{attribute 'qualified_only'}
{attribute 'to_string'}
// ------------------------------------------------------------------------- 
//  SRCI Robot Library                                                
// ------------------------------------------------------------------------- 
//                                                                           
//  Object:      SyncReaction                                       
//  Author:      Thorsten Brach                                                
//  Date:        2024-06-01
//
//  Description:                                              
//   
//                                                                           
//  Copyright: 
//    (C) 2024 Thorsten Brach. All rights reserved                                                                                                                                            
//             Licensed under the MIT License.
//                                                                           
//  Disclaimer:                                                                           
//    This project is provided without any guarantee and can be used for   
//    private and commercial purposes. Any use is at the user’s 
//    own risk and responsibility.
//
// -------------------------------------------------------------------------
TYPE SyncReaction :
(
  /// • System behavior unaffected
  NO_REACTION := 0,
  /// • No automatic disable
  /// • Reaction will only apply when RA is disabled
  /// • RA can only be enabled if client and server are synchronized
  NO_AUTOMATIC_DISABLE := 1,  
  /// • No automatic disable
  /// • RA can only be enabled if client and server are synchronized
  /// • RA sequence state will change to interrupted when no command is buffered in the active sequence
  /// • Continuation is only possible if client and server are synchronized
  INTERRUPT_WHEN_SEQUENCE_IS_EMPTY := 2,  
  /// • No automatic disable
  /// • RA can only be enabled if client and server are synchronized
  /// • RA sequence state will change to interrupted
  /// • Continuation is only possible if client and server are synchronized
  IMMEDIATE_INTERRUPT := 3
)USINT;
END_TYPE

{attribute 'qualified_only'}
{attribute 'to_string'}
// ------------------------------------------------------------------------- 
//  SRCI Robot Library                                                
// ------------------------------------------------------------------------- 
//                                                                           
//  Object:      SyncTime                                       
//  Author:      Thorsten Brach                                                
//  Date:        2025-04-13
//
//  Description:                                              
//   
//                                                                           
//  Copyright: 
//    (C) 2025 Thorsten Brach. All rights reserved                                                                                                                                            
//             Licensed under the MIT License.
//                                                                           
//  Disclaimer:                                                                           
//    This project is provided without any guarantee and can be used for   
//    private and commercial purposes. Any use is at the user’s 
//    own risk and responsibility.
//
// -------------------------------------------------------------------------
TYPE SyncTime :
(
  /// Synchronization during startup
	DURING_START_UP := 0,
  /// Synchronization after startup
  AFTER_START_UP := 1
)DINT;
END_TYPE

{attribute 'qualified_only'}
{attribute 'to_string'}
// ------------------------------------------------------------------------- 
//  SRCI Robot Library                                                
// ------------------------------------------------------------------------- 
//                                                                           
//  Object:      TriggerCondition                                       
//  Author:      Thorsten Brach                                                
//  Date:        2024-06-01
//
//  Description:                                              
//   
//                                                                           
//  Copyright: 
//    (C) 2024 Thorsten Brach. All rights reserved                                                                                                                                            
//             Licensed under the MIT License.
//                                                                           
//  Disclaimer:                                                                           
//    This project is provided without any guarantee and can be used for   
//    private and commercial purposes. Any use is at the user’s 
//    own risk and responsibility.
//
// -------------------------------------------------------------------------
TYPE TriggerCondition :
(
  /// 5: Time in ms  - point reference is target position
  TARGET_POSITION_TIME_MS := -5,
  /// 4: TCP velocity in mm/s - point reference is target position
  TARGET_POSITION_TCP_VELOCITY_ABSOLUTE := -4,
  /// 3: TCP velocity in % of reference velocity - point reference is target position
  TARGET_POSITION_TCP_VELOCITY_PERCENT := -3,
  /// 2: Distance in mm of trajectory - point reference is target position
  TARGET_POSITION_DISTANCE_ABSOLUTE := -2,
  /// 1: Distance in % of trajectory - point reference is target position
  TARGET_POSITION_DISTANCE_PERCENT := -1,
  /// 0: Undfined 
  UNDEFINED := 0,
  /// 1: Distance in % of trajectory - point reference is start position
  START_POSITION_DISTANCE_PERCENT := 1,
  /// 2: Distance in mm of trajectory - point reference is start position
  START_POSITION_DISTANCE_ABSOLUTE := 2,
  /// 3: TCP velocity in % of reference velocity - point reference is start position
  START_POSITION_TCP_VELOCITY_PERCENT := 3,
  /// 4: TCP velocity in mm/s - point reference is start position
  START_POSITION_TCP_VELOCIT_ABSOLUTE := 4,
  /// 5: Time in ms - point reference is start position
  START_POSITION_TIME_MS := 5
)SINT;
END_TYPE

{attribute 'qualified_only'}
{attribute 'to_string'}
// ------------------------------------------------------------------------- 
//  SRCI Robot Library                                                
// ------------------------------------------------------------------------- 
//                                                                           
//  Object:      UnitLimitAxis                                       
//  Author:      Thorsten Brach                                                
//  Date:        2025-02-23
//
//  Description:                                              
//   
//                                                                           
//  Copyright: 
//    (C) 2025 Thorsten Brach. All rights reserved                                                                                                                                            
//             Licensed under the MIT License.
//                                                                           
//  Disclaimer:                                                                           
//    This project is provided without any guarantee and can be used for   
//    private and commercial purposes. Any use is at the user’s 
//    own risk and responsibility.
//
// -------------------------------------------------------------------------

TYPE UnitLimitAxis :
(
  /// Percentage (%) (default)
	PERCENTAGE  := 0,
  /// Newton meter (Nm)
  NEWTONMETER := 1,
  /// Milliampere (mA)
  MILLIAMPERE := 2  
)USINT;
END_TYPE

{attribute 'qualified_only'}
{attribute 'to_string'}
// ------------------------------------------------------------------------- 
//  SRCI Robot Library                                                
// ------------------------------------------------------------------------- 
//                                                                           
//  Object:      AbortingMode                                       
//  Author:      Thorsten Brach                                                
//  Date:        2024-06-01
//
//  Description:                                              
//   
//                                                                           
//  Copyright: 
//    (C) 2024 Thorsten Brach. All rights reserved                                                                                                                                            
//             Licensed under the MIT License.
//                                                                           
//  Disclaimer:                                                                           
//    This project is provided without any guarantee and can be used for   
//    private and commercial purposes. Any use is at the user’s 
//    own risk and responsibility.
//
// -------------------------------------------------------------------------
TYPE AbortingMode :
(
  /// The current movement command as well as all stored movements are executed as programmed. 
  /// The new motion command is queued in the motion buffer.
  BUFFER := 0,
  /// The current movement command is aborted. All buffered motion movements are discarded. 
  /// The new target position is approached, depending on the motion command.
  ABORT  := 1
)SINT;
END_TYPE

TYPE AbortingModeEnum : AbortingMode; END_TYPE;

{attribute 'qualified_only'}
{attribute 'to_string'}
// ------------------------------------------------------------------------- 
//  SRCI Robot Library                                                
// ------------------------------------------------------------------------- 
//                                                                           
//  Object:      BlendingMode                                       
//  Author:      Thorsten Brach                                                
//  Date:        2024-06-01
//
//  Description:                                              
//   
//                                                                           
//  Copyright: 
//    (C) 2024 Thorsten Brach. All rights reserved                                                                                                                                            
//             Licensed under the MIT License.
//                                                                           
//  Disclaimer:                                                                           
//    This project is provided without any guarantee and can be used for   
//    private and commercial purposes. Any use is at the user’s 
//    own risk and responsibility.
//
// -------------------------------------------------------------------------
TYPE BlendingMode :
(
  /// Appended, buffered, no blending
  EXACT_STOP := 0,
  /// Start blending when the defined velocity is reached
  DEFINED_VELOCITY := 2,
  /// Define blending sphere with radius
  CORNER_DISTANCE := 3,
  /// Define blending with deviation
  MAX_CORNER_DEVIATION := 4,
  /// Define blending sphere with 2 radiuses
  CORNER_DISTANCE_2R := 10,
  /// Define blending with percentage of overlapping of deceleration and acceleration ramp
  RAMP_OVERLAP := 11,
  /// Define blending sphere with starting radius
  CORNER_DISTANCE_1R := 12
)USINT;
END_TYPE

{attribute 'qualified_only'}
{attribute 'to_string'}
// ------------------------------------------------------------------------- 
//  SRCI Robot Library                                                
// ------------------------------------------------------------------------- 
//                                                                           
//  Object:      CircMode                                       
//  Author:      Thorsten Brach                                                
//  Date:        2024-06-01
//
//  Description:                                              
//   
//                                                                           
//  Copyright: 
//    (C) 2024 Thorsten Brach. All rights reserved                                                                                                                                            
//             Licensed under the MIT License.
//                                                                           
//  Disclaimer:                                                                           
//    This project is provided without any guarantee and can be used for   
//    private and commercial purposes. Any use is at the user’s 
//    own risk and responsibility.
//
// -------------------------------------------------------------------------
TYPE CircMode :
(
  /// "AuxPoint" defines a point on the circle crossed on the path from the starting to the end point.
  BORDER := 0,
  /// "AuxPoint" defines the center point of the circle.
  CENTER := 1,
  /// "AuxPoint" defines the center point of the circle, "Angle" defines the end position of the circular motion, and "CircPlane" defines the circle’s plane.
  CENTER_WITH_ANGLE := 2,
  /// "AuxPoint" defines a vector which length is the radius of the circle. The plane of the circle is defined by the rule of right thumb while the "AuxPoint" defines the spearhead point of the perpendicular.
  RADIUS := 3
)SINT;
END_TYPE

{attribute 'qualified_only'}
{attribute 'to_string'}
// ------------------------------------------------------------------------- 
//  SRCI Robot Library                                                
// ------------------------------------------------------------------------- 
//                                                                           
//  Object:      CollisionReactionMode                                       
//  Author:      Thorsten Brach                                                
//  Date:        2024-06-01
//
//  Description:                                              
//   
//                                                                           
//  Copyright: 
//    (C) 2024 Thorsten Brach. All rights reserved                                                                                                                                            
//             Licensed under the MIT License.
//                                                                           
//  Disclaimer:                                                                           
//    This project is provided without any guarantee and can be used for   
//    private and commercial purposes. Any use is at the user’s 
//    own risk and responsibility.
//
// -------------------------------------------------------------------------
TYPE CollisionReactionMode :
(
  /// Standing still
  STANDING_STILL := 0,
  /// Reversed movement
  REVERSED_MOVEMENT := 1
)USINT;
END_TYPE

{attribute 'qualified_only'}
{attribute 'to_string'}
// ------------------------------------------------------------------------- 
//  SRCI Robot Library                                                
// ------------------------------------------------------------------------- 
//                                                                           
//  Object:      ConnectionMode                                       
//  Author:      Thorsten Brach                                                
//  Date:        2024-06-01
//
//  Description:                                              
//   
//                                                                           
//  Copyright: 
//    (C) 2024 Thorsten Brach. All rights reserved                                                                                                                                            
//             Licensed under the MIT License.
//                                                                           
//  Disclaimer:                                                                           
//    This project is provided without any guarantee and can be used for   
//    private and commercial purposes. Any use is at the user’s 
//    own risk and responsibility.
//
// -------------------------------------------------------------------------
TYPE ConnectionMode :
(
  /// Encoder is connected to RC
  RC_CONNECTED := 0,
  /// Encoder is connected to PLC
  PLC_CONNECTED := 1
)SINT;
END_TYPE

{attribute 'qualified_only'}
{attribute 'to_string'}
// ------------------------------------------------------------------------- 
//  SRCI Robot Library                                                
// ------------------------------------------------------------------------- 
//                                                                           
//  Object:      DefinitionMode                                       
//  Author:      Thorsten Brach                                                
//  Date:        2024-06-01
//
//  Description:                                              
//   
//                                                                           
//  Copyright: 
//    (C) 2024 Thorsten Brach. All rights reserved                                                                                                                                            
//             Licensed under the MIT License.
//                                                                           
//  Disclaimer:                                                                           
//    This project is provided without any guarantee and can be used for   
//    private and commercial purposes. Any use is at the user’s 
//    own risk and responsibility.
//
// -------------------------------------------------------------------------
TYPE DefinitionMode :
(
  /// ZeroPoint describes center point of body 
  Center := 1,
  /// ZeroPoint describes point on face of body. Parameter values for X2, Y2, Z2 will be ignored  
  Face := 2 
)USINT;
END_TYPE

{attribute 'qualified_only'}
{attribute 'to_string'}
// ------------------------------------------------------------------------- 
//  SRCI Robot Library                                                
// ------------------------------------------------------------------------- 
//                                                                           
//  Object:      DetectionMode                                       
//  Author:      Thorsten Brach                                                
//  Date:        2024-06-01
//
//  Description:                                              
//   
//                                                                           
//  Copyright: 
//    (C) 2024 Thorsten Brach. All rights reserved                                                                                                                                            
//             Licensed under the MIT License.
//                                                                           
//  Disclaimer:                                                                           
//    This project is provided without any guarantee and can be used for   
//    private and commercial purposes. Any use is at the user’s 
//    own risk and responsibility.
//
// -------------------------------------------------------------------------
TYPE DetectionMode :
(
  /// Torque (default)
  TORQUE := 0,
  /// Force
  FORCE := 1,
  /// Electrical current
  ELECTRICAL_CURRENT := 2,
  /// Following Error
  FOLLOWING_ERROR := 3
)USINT;
END_TYPE

{attribute 'qualified_only'}
{attribute 'to_string'}
// ------------------------------------------------------------------------- 
//  SRCI Robot Library                                                
// ------------------------------------------------------------------------- 
//                                                                           
//  Object:      ErrorTriggerMode                                       
//  Author:      Thorsten Brach                                                
//  Date:        2024-06-01
//
//  Description:                                              
//   
//                                                                           
//  Copyright: 
//    (C) 2024 Thorsten Brach. All rights reserved                                                                                                                                            
//             Licensed under the MIT License.
//                                                                           
//  Disclaimer:                                                                           
//    This project is provided without any guarantee and can be used for   
//    private and commercial purposes. Any use is at the user’s 
//    own risk and responsibility.
//
// -------------------------------------------------------------------------
TYPE ErrorTriggerMode :
(
  /// Any command (default)
  ANY_COMMAND := 0,
  /// General commands
  GENERAL_COMMANDS := 1,
  /// Administrative commands
  ADMINISTRATIVE_COMMANDS := 2,
  /// Move commands
  MOVE_COMMANDS := 3,
  /// Periphery commands
  PERIPHERY_COMMANDS := 4,
  /// Extended commands
  EXTENDED_COMMANDS := 5,
  /// Specific command or RI message
  SPECIFIC_COMMAND_OR_RI_MESSAGE := 6,
  /// Specific RC or RA message code
  SPECIFIC_RC_OR_RA_MESSAGE_CODE := 7,
  /// Any RI message code
  ANY_RI_MESSAGE_CODE := 8,
  /// Any RC or RA message code
  ANY_RC_OR_RA_MESSAGE_CODE := 9
)SINT;
END_TYPE

{attribute 'qualified_only'}
{attribute 'to_string'}
// ------------------------------------------------------------------------- 
//  SRCI Robot Library                                                
// ------------------------------------------------------------------------- 
//                                                                           
//  Object:      ExecutionMode                                       
//  Author:      Thorsten Brach                                                
//  Date:        2024-06-01
//
//  Description:                                              
//   
//                                                                           
//  Copyright: 
//    (C) 2024 Thorsten Brach. All rights reserved                                                                                                                                            
//             Licensed under the MIT License.
//                                                                           
//  Disclaimer:                                                                           
//    This project is provided without any guarantee and can be used for   
//    private and commercial purposes. Any use is at the user’s 
//    own risk and responsibility.
//
// -------------------------------------------------------------------------
TYPE ExecutionMode :
(
  /// Command is buffered in sequence buffer and executed once
  SEQUENCE_PRIMARY := 0,
  /// Command is buffered in sequence buffer, aborts and empties previous commands in sequence buffer, and is executed once
  SEQUENCE_ABORT_OTHERS_PRIMARY := 1,
  /// Command is buffered in parallel buffer and executed once. The execution may also be Trigger based.
  PARALLEL := 2,
  /// Command is buffered in parallel buffer and executed repeatedly until deliberate deactivation by user. The de- and activation may also be Trigger based.
  CONTINUOUS := 3,
  /// Command is buffered and executed once when triggered. The CMD remains in the buffer until removed by the user.
  TRIGGER_MULTIPLE := 5,
  /// Command is buffered in sequence buffer and executed once (Secondary)
  SEQUENCE_SECONDARY := 7,
  /// Command is buffered in sequence buffer, aborts and empties previous commands in sequence buffer and is executed once (Secondary)
  SEQUENCE_ABORT_OTHERS_SECONDARY := 8,
  /// CMD execution is stopped and/or CMD is removed from the buffer.
  STOP_PARALLEL_CONTINUOUS_TRIGGER := 9
)USINT;
END_TYPE

{attribute 'qualified_only'}
{attribute 'to_string'}
// ------------------------------------------------------------------------- 
//  SRCI Robot Library                                                
// ------------------------------------------------------------------------- 
//                                                                           
//  Object:      FrameCalculationMode                                       
//  Author:      Thorsten Brach                                                
//  Date:        2024-06-01
//
//  Description:                                              
//   
//                                                                           
//  Copyright: 
//    (C) 2024 Thorsten Brach. All rights reserved                                                                                                                                            
//             Licensed under the MIT License.
//                                                                           
//  Disclaimer:                                                                           
//    This project is provided without any guarantee and can be used for   
//    private and commercial purposes. Any use is at the user’s 
//    own risk and responsibility.
//
// -------------------------------------------------------------------------
TYPE FrameCalculationMode :
(
  /// 0: Three-Point-method (default)
  THREE_POINT_METHOD := 0,  
  /// 1: Four-Point-method
  FOUR_POINT_METHOD := 1,  
  /// 2: One-Point-method
  ONE_POINT_METHOD := 2
)SINT;
END_TYPE

{attribute 'qualified_only'}
{attribute 'to_string'}
// ------------------------------------------------------------------------- 
//  SRCI Robot Library                                                
// ------------------------------------------------------------------------- 
//                                                                           
//  Object:      FunctionMode                                       
//  Author:      Thorsten Brach                                                
//  Date:        2024-06-01
//
//  Description:                                              
//   
//                                                                           
//  Copyright: 
//    (C) 2024 Thorsten Brach. All rights reserved                                                                                                                                            
//             Licensed under the MIT License.
//                                                                           
//  Disclaimer:                                                                           
//    This project is provided without any guarantee and can be used for   
//    private and commercial purposes. Any use is at the user’s 
//    own risk and responsibility.
//
// -------------------------------------------------------------------------
TYPE FunctionMode :
(
  enum_member := 0
);
END_TYPE

{attribute 'qualified_only'}
{attribute 'to_string'}
// ------------------------------------------------------------------------- 
//  SRCI Robot Library                                                
// ------------------------------------------------------------------------- 
//                                                                           
//  Object:      InterpolationMode                                       
//  Author:      Thorsten Brach                                                
//  Date:        2024-06-01
//
//  Description:                                              
//   
//                                                                           
//  Copyright: 
//    (C) 2024 Thorsten Brach. All rights reserved                                                                                                                                            
//             Licensed under the MIT License.
//                                                                           
//  Disclaimer:                                                                           
//    This project is provided without any guarantee and can be used for   
//    private and commercial purposes. Any use is at the user’s 
//    own risk and responsibility.
//
// -------------------------------------------------------------------------
TYPE InterpolationMode :
(
  /// Linear interpolation
  Linear_interpolation := 0,
  /// Direct interpolation (PTP)
  Direct_interpolation := 1
)USINT;
END_TYPE

{attribute 'qualified_only'}
{attribute 'to_string'}
// ------------------------------------------------------------------------- 
//  SRCI Robot Library                                                
// ------------------------------------------------------------------------- 
//                                                                           
//  Object:      JogMode                                       
//  Author:      Thorsten Brach                                                
//  Date:        2024-06-01
//
//  Description:                                              
//   
//                                                                           
//  Copyright: 
//    (C) 2024 Thorsten Brach. All rights reserved                                                                                                                                            
//             Licensed under the MIT License.
//                                                                           
//  Disclaimer:                                                                           
//    This project is provided without any guarantee and can be used for   
//    private and commercial purposes. Any use is at the user’s 
//    own risk and responsibility.
//
// -------------------------------------------------------------------------
TYPE JogMode :
(
  /// • Jog TCP manually in the given frame (WCS/UCS)
  /// • Movement on several coordinate axes simultaneously possible
  JOG_FRAME := 0,
  /// • Jog TCP manually in the given tool coordinate system
  /// • Movement on several coordinate axes simultaneously possible
  JOG_TOOL := 1,
  /// • Jog joints manually without referring to a given frame or tool
  /// • Movement of several axes simultaneously possible.
  JOG_AXES := 2
)USINT;
END_TYPE

{attribute 'qualified_only'}
{attribute 'to_string'}
// ------------------------------------------------------------------------- 
//  SRCI Robot Library                                                
// ------------------------------------------------------------------------- 
//                                                                           
//  Object:      LimitMode                                       
//  Author:      Thorsten Brach                                                
//  Date:        2024-06-01
//
//  Description:                                              
//   
//                                                                           
//  Copyright: 
//    (C) 2024 Thorsten Brach. All rights reserved                                                                                                                                            
//             Licensed under the MIT License.
//                                                                           
//  Disclaimer:                                                                           
//    This project is provided without any guarantee and can be used for   
//    private and commercial purposes. Any use is at the user’s 
//    own risk and responsibility.
//
// -------------------------------------------------------------------------
TYPE LimitMode :
(
  /// 0: No limit defined (default)
  /// The robot can be moved in the direction set with the input parameter "CompliantAxes" in a compliant manner by applying an external force on it.
  /// By reaching the mechanical or software limits, the robot stops.
  NO_LIMIT_DEFINED := 0,
  
  /// 1: Limit defined
  /// The robot can be moved along the defined vector in a compliant manner by applying an external force on it.
  /// By reaching the vector limit defined by the input parameter "VectorData", the robot stops.
  LIMIT_DEFINED := 1
)USINT;
END_TYPE

{attribute 'qualified_only'}
{attribute 'to_string'}
// ------------------------------------------------------------------------- 
//  SRCI Robot Library                                                
// ------------------------------------------------------------------------- 
//                                                                           
//  Object:      LoadMeasurementMode                                       
//  Author:      Thorsten Brach                                                
//  Date:        2024-06-01
//
//  Description:                                              
//   
//                                                                           
//  Copyright: 
//    (C) 2024 Thorsten Brach. All rights reserved                                                                                                                                            
//             Licensed under the MIT License.
//                                                                           
//  Disclaimer:                                                                           
//    This project is provided without any guarantee and can be used for   
//    private and commercial purposes. Any use is at the user’s 
//    own risk and responsibility.
//
// -------------------------------------------------------------------------
TYPE  LoadMeasurementMode :
(
  /// 0: One Position (default)
  /// Use one defined position and optional axes ranges
  ONE_POSITION := 0,  
  /// 1: Configuration Angle
  /// Use one defined position and optional axes ranges
  CONFIGURATION_ANGLE := 1,  
  /// 2: Area
  /// Use a defined area for the measurement
  AREA := 2,  
  /// 3: Two Positions
  /// Use defined positions for the measurement
  TWO_POSITIONS := 3
)USINT;
END_TYPE

{attribute 'qualified_only'}
{attribute 'to_string'}
// ------------------------------------------------------------------------- 
//  SRCI Robot Library                                                
// ------------------------------------------------------------------------- 
//                                                                           
//  Object:      LogonMode                                       
//  Author:      Thorsten Brach                                                
//  Date:        2024-06-01
//
//  Description:                                              
//   
//                                                                           
//  Copyright: 
//    (C) 2024 Thorsten Brach. All rights reserved                                                                                                                                            
//             Licensed under the MIT License.
//                                                                           
//  Disclaimer:                                                                           
//    This project is provided without any guarantee and can be used for   
//    private and commercial purposes. Any use is at the user’s 
//    own risk and responsibility.
//
// -------------------------------------------------------------------------
TYPE LogonMode :
(
  /// Password only (default)
  PASSWORD_ONLY := 0,
  /// Username and Password
  USERNAME_AND_PASSWORD := 1,
  /// Level ID and Password
  LEVEL_ID_AND_PASSWORD := 2
)SINT;
END_TYPE

{attribute 'qualified_only'}
{attribute 'to_string'}
// ------------------------------------------------------------------------- 
//  SRCI Robot Library                                                
// ------------------------------------------------------------------------- 
//                                                                           
//  Object:      MeasuringIoMode                                       
//  Author:      Thorsten Brach                                                
//  Date:        2024-06-01
//
//  Description:                                              
//   
//                                                                           
//  Copyright: 
//    (C) 2024 Thorsten Brach. All rights reserved                                                                                                                                            
//             Licensed under the MIT License.
//                                                                           
//  Disclaimer:                                                                           
//    This project is provided without any guarantee and can be used for   
//    private and commercial purposes. Any use is at the user’s 
//    own risk and responsibility.
//
// -------------------------------------------------------------------------
TYPE MeasuringIoMode :
(
  /// Measurement at next rising edge 
  /// • Output "MeasuredPosition_1" used
  MEASUREMENT_AT_NEXT_RISING_EDGE := 0,
  /// Measurement at next falling edge 
  /// • Output "MeasuredPosition_1" used
  MEASUREMENT_AT_NEXT_FALLING_EDGE := 1,
  /// Measurement at next edges, regardless of rising or falling edges.
  /// • First position stored in output "MeasuredPosition_1"
  /// • Second position stored in output "MeasuredPosition_2"
  MEASUREMENT_AT_NEXT_EDGE := 2,
  /// Measurement at two edges, beginning with the rising edge:
  /// • Rising edge = "MeasuredPosition_1 "
  /// • Falling edge = "MeasuredPosition_2 "
  MEASUREMENT_AT_TWO_EDGES_BEGIN_WITH_RISING := 3,
  /// Measurement at two edges, beginning with the falling edge:
  /// • Falling edge = " MeasuredPosition_1 "
  /// • Rising edge = "MeasuredPosition_2 "
  MEASUREMENT_AT_TWO_EDGES_BEGIN_WITH_FALLING := 4
)USINT;
END_TYPE

{attribute 'qualified_only'}
{attribute 'to_string'}
// ------------------------------------------------------------------------- 
//  SRCI Robot Library                                                
// ------------------------------------------------------------------------- 
//                                                                           
//  Object:      MeasuringUnitMode                                       
//  Author:      Thorsten Brach                                                
//  Date:        2024-06-01
//
//  Description:                                              
//   
//                                                                           
//  Copyright: 
//    (C) 2024 Thorsten Brach. All rights reserved                                                                                                                                            
//             Licensed under the MIT License.
//                                                                           
//  Disclaimer:                                                                           
//    This project is provided without any guarantee and can be used for   
//    private and commercial purposes. Any use is at the user’s 
//    own risk and responsibility.
//
// -------------------------------------------------------------------------
TYPE MeasuringUnitMode :
(
  /// 0: VectorLength (default)
  ///    Defines the distance in millimeter between two points in cartesian space.
  VECTOR_LENGTH  := 0,
  /// 1: SegmentLength
  ///    Defines the distance in mm covered between the two points in cartesian space
  SEGMENT_LENGTH := 1,
  /// 2: Time
  ///    Defines the duration in milliseconds between the start and end point.
  TIME_DURATION  := 2
)USINT;
END_TYPE

{attribute 'qualified_only'}
{attribute 'to_string'}
// ------------------------------------------------------------------------- 
//  SRCI Robot Library                                                
// ------------------------------------------------------------------------- 
//                                                                           
//  Object:      OperationMode                                       
//  Author:      Thorsten Brach                                                
//  Date:        2024-06-01
//
//  Description:                                              
//   
//                                                                           
//  Copyright: 
//    (C) 2024 Thorsten Brach. All rights reserved                                                                                                                                            
//             Licensed under the MIT License.
//                                                                           
//  Disclaimer:                                                                           
//    This project is provided without any guarantee and can be used for   
//    private and commercial purposes. Any use is at the user’s 
//    own risk and responsibility.
//
// -------------------------------------------------------------------------
TYPE OperationMode :
(
 /// Test mode 1:
 /// • Maximum velocity of TCP is restricted to <250 mm/s
 /// • Robot can only be moved while enable switch is active
 /// • Designed for jogging, teaching program, verification
 /// • Safety door can be opened
 T1_LOCAL := 1,
 /// Test mode 2:
 /// • Maximum velocity of TCP not restricted (100%)
 /// • Robot can only be moved while enable switch is active
 /// • Designed for program verification (step mode)
 /// • Safety door can be opened
 T2_LOCAL := 2,
 /// Automatic mode:
 /// • Maximum velocity of TCP not restricted (100%)
 /// • Robot is executing user program automatically
 /// • Robot will stop if safety devices report error (e.g. safety door must be closed)
 AUTO := 3,
 /// External Automatic mode (PLC mode)
 /// • Robot is operated remotely only
 /// • Maximum velocity of TCP not restricted (100%)
 /// • Robot is executing user program automatically
 /// • Jogging possible
 /// • Robot will stop if safety devices report error (e.g. safety door must be closed)
 AUTO_EXT := 4,
 /// External Test mode 1 (PLC mode with T1 functionality)
 /// • Robot is operated remotely only
 /// • Maximum velocity of TCP is restricted to <250 mm/s
 /// • Robot can only be moved while enable switch is active
 /// • Designed for jogging, teaching, program verification
 /// • Safety door can be opened
 T1_EXT := 5,
 /// External Test mode 2:
 /// • Robot is operated remotely only
 /// • Maximum velocity of TCP not restricted (100%)
 /// • Robot can only be moved while enable switch is active
 /// • Designed for jogging, program verification (step mode)
 /// • Safety door can be opened
 T2_EXT := 6
)USINT;
END_TYPE

{attribute 'qualified_only'}
{attribute 'to_string'}
// ------------------------------------------------------------------------- 
//  SRCI Robot Library                                                
// ------------------------------------------------------------------------- 
//                                                                           
//  Object:      OrientationMode                                       
//  Author:      Thorsten Brach                                                
//  Date:        2024-06-01
//
//  Description:                                              
//   
//                                                                           
//  Copyright: 
//    (C) 2024 Thorsten Brach. All rights reserved                                                                                                                                            
//             Licensed under the MIT License.
//                                                                           
//  Disclaimer:                                                                           
//    This project is provided without any guarantee and can be used for   
//    private and commercial purposes. Any use is at the user’s 
//    own risk and responsibility.
//
// -------------------------------------------------------------------------
TYPE OrientationMode :
(
    /// Change orientation continuously in a linear way
    LINEAR_INTERPOLATED := 1,
    /// Change orientation continuously in a joint interpolated way of wrist joints
    JOINT_INTERPOLATED := 2,
    /// No change of orientation during movement
    FIX := 3,
    /// No change of orientation in relation to trajectory
    PATH := 4
)SINT;
END_TYPE

{attribute 'qualified_only'}
{attribute 'to_string'}
// ------------------------------------------------------------------------- 
//  SRCI Robot Library                                                
// ------------------------------------------------------------------------- 
//                                                                           
//  Object:      OriMode                                       
//  Author:      Thorsten Brach                                                
//  Date:        2024-06-01
//
//  Description:                                              
//   
//                                                                           
//  Copyright: 
//    (C) 2024 Thorsten Brach. All rights reserved                                                                                                                                            
//             Licensed under the MIT License.
//                                                                           
//  Disclaimer:                                                                           
//    This project is provided without any guarantee and can be used for   
//    private and commercial purposes. Any use is at the user’s 
//    own risk and responsibility.
//
// -------------------------------------------------------------------------
TYPE OriMode :
(
  /// Change orientation continuously in a linear way
  LINEAR_INTERPOLATED := 1,
  /// Change orientation continuously in a joint interpolated way.
  JOINT_INTERPOLATED  := 2,
  /// No change of orientation during movement
  FIX                 := 3,
  /// No change of orientation in relation to trajectory
  PATH                := 4
)USINT;
END_TYPE

{attribute 'qualified_only'}
{attribute 'to_string'}
// ------------------------------------------------------------------------- 
//  SRCI Robot Library                                                
// ------------------------------------------------------------------------- 
//                                                                           
//  Object:      ProcessingMode                                       
//  Author:      Thorsten Brach                                                
//  Date:        2024-06-01
//
//  Description:                                              
//   
//                                                                           
//  Copyright: 
//    (C) 2024 Thorsten Brach. All rights reserved                                                                                                                                            
//             Licensed under the MIT License.
//                                                                           
//  Disclaimer:                                                                           
//    This project is provided without any guarantee and can be used for   
//    private and commercial purposes. Any use is at the user’s 
//    own risk and responsibility.
//
// -------------------------------------------------------------------------
TYPE ProcessingMode :
(
  /// Command is buffered in sequence buffer and executed once
  BUFFERED := 0,
  /// Command is buffered in sequence buffer, aborts and empties previous commands in sequence buffer, and is executed once
  ABORTING := 1,
  /// Command is buffered in parallel buffer and executed once
  PARALLEL := 2,
  /// Command is buffered in parallel buffer and executed repeatedly until deliberate deactivation by user
  CONTINUOUS := 3,
  /// CMD execution is stopped and/or CMD is removed from the buffer
  DEACTIVATE := 9,
  /// Command is buffered in sequence buffer and executed once (Trigger based)
  TRIGGER_BUFFERED := 10,
  /// Command is buffered in sequence buffer, aborts and empties previous commands in sequence buffer, and is executed once (Trigger based)
  TRIGGER_ABORTING := 11,
  /// Command is buffered in parallel buffer and executed once (Trigger based)
  TRIGGER_ONCE := 12,
  /// Command is buffered in parallel buffer and executed repeatedly until deliberate deactivation by user (Trigger based)
  TRIGGER_CONTINUOUS := 13,
  /// Command is buffered and executed multiple times when triggered. The CMD remains in the buffer until removed by the user.
  TRIGGER_MULTIPLE := 14
)USINT;
END_TYPE

TYPE ProcessingModeEnum : ProcessingMode; END_TYPE

{attribute 'qualified_only'}
{attribute 'to_string'}
// ------------------------------------------------------------------------- 
//  SRCI Robot Library                                                
// ------------------------------------------------------------------------- 
//                                                                           
//  Object:      ResistanceForceMode                                       
//  Author:      Thorsten Brach                                                
//  Date:        2024-06-01
//
//  Description:                                              
//   
//                                                                           
//  Copyright: 
//    (C) 2024 Thorsten Brach. All rights reserved                                                                                                                                            
//             Licensed under the MIT License.
//                                                                           
//  Disclaimer:                                                                           
//    This project is provided without any guarantee and can be used for   
//    private and commercial purposes. Any use is at the user’s 
//    own risk and responsibility.
//
// -------------------------------------------------------------------------
TYPE ResistanceForceMode :
(
  /// 0 (default): ResistanceForceTCP.
  /// Set "0" to set the resistance of the RA against the external force at the TCP.
  RESISTANCE_FORCE_TCP := 0,
  
  /// 1: ResistanceForceAxis.
  /// Set "1" to set the resistance of the RA against the external force for each axis independently.
  RESISTANCE_FORCE_AXIS := 1
)USINT;
END_TYPE

{attribute 'qualified_only'}
TYPE ReturnMode :
(
  /// Interrupt position
  INTERRUPT_POSITION := 0,
  /// End position
  END_POSITION := 1
)BYTE;
END_TYPE

{attribute 'qualified_only'}
// ------------------------------------------------------------------------- 
//  SRCI Robot Library                                                
// ------------------------------------------------------------------------- 
//                                                                           
//  Object:      SensorConnectionMode                                       
//  Author:      Thorsten Brach                                                
//  Date:        2024-06-01
//
//  Description:                                              
//   
//                                                                           
//  Copyright: 
//    (C) 2024 Thorsten Brach. All rights reserved                                                                                                                                            
//             Licensed under the MIT License.
//                                                                           
//  Disclaimer:                                                                           
//    This project is provided without any guarantee and can be used for   
//    private and commercial purposes. Any use is at the user’s 
//    own risk and responsibility.
//
// -------------------------------------------------------------------------
TYPE SensorConnectionMode :
(
  /// RC sensor and algorithm
  /// Force-Torque-Sensor connected to RC
  /// Control algorithm in RC
  RC_SENSOR_ALGORITHM := 0,
  
  /// PLC sensor and RC algorithm
  /// Force-Torque-Sensor connected to PLC
  /// Control algorithm in RC
  PLC_SENSOR_RC_ALGORITHM := 1,
  
  /// PLC sensor and algorithm
  /// Force-Torque-Sensor connected to PLC
  /// Control algorithm in PLC
  PLC_SENSOR_ALGORITHM := 2
)USINT;
END_TYPE

{attribute 'qualified_only'}
// ------------------------------------------------------------------------- 
//  SRCI Robot Library                                                
// ------------------------------------------------------------------------- 
//                                                                           
//  Object:      SingularityAvoidanceMode                                       
//  Author:      Thorsten Brach                                                
//  Date:        2024-06-01
//
//  Description:                                              
//   
//                                                                           
//  Copyright: 
//    (C) 2024 Thorsten Brach. All rights reserved                                                                                                                                            
//             Licensed under the MIT License.
//                                                                           
//  Disclaimer:                                                                           
//    This project is provided without any guarantee and can be used for   
//    private and commercial purposes. Any use is at the user’s 
//    own risk and responsibility.
//
// -------------------------------------------------------------------------
TYPE SingularityAvoidanceMode :
(
  /// 0: NoChange (default)
  /// Allow movement of one or more joints to avoid singularities without a change of the orientation
  NO_CHANGE := 0,
  
  /// 1: Lock J4
  /// Lock the 4th joint to avoid singularities
  LOCK_J4 := 1,
  
  /// 2: ToolOrientation
  /// Allow a small movement of the tool orientation to avoid singularities
  TOOL_ORIENTATION := 2
)USINT;
END_TYPE

{attribute 'qualified_only'}
// ------------------------------------------------------------------------- 
//  SRCI Robot Library                                                
// ------------------------------------------------------------------------- 
//                                                                           
//  Object:      SplineMode                                       
//  Author:      Thorsten Brach                                                
//  Date:        2024-06-01
//
//  Description:                                              
//   
//                                                                           
//  Copyright: 
//    (C) 2024 Thorsten Brach. All rights reserved                                                                                                                                            
//             Licensed under the MIT License.
//                                                                           
//  Disclaimer:                                                                           
//    This project is provided without any guarantee and can be used for   
//    private and commercial purposes. Any use is at the user’s 
//    own risk and responsibility.
//
// -------------------------------------------------------------------------
TYPE SplineMode :
(
  /// 0: Discrete Points
  DISCRETE_POINTS := 0,
  /// 1: Bézier Spline
  BEZIER_SPLINE := 1,
  /// 2: B-Splines
  B_SPLINES := 2,
  /// 3: Cubic Hermite Spline
  CUBIC_HERMITE_SPLINE := 3,
  /// 4: C-Splines
  C_SPLINES := 4
)UINT;
END_TYPE

{attribute 'qualified_only'}
// ------------------------------------------------------------------------- 
//  SRCI Robot Library                                                
// ------------------------------------------------------------------------- 
//                                                                           
//  Object:      StepMode                                       
//  Author:      Thorsten Brach                                                
//  Date:        2024-06-01
//
//  Description:                                              
//   
//                                                                           
//  Copyright: 
//    (C) 2024 Thorsten Brach. All rights reserved                                                                                                                                            
//             Licensed under the MIT License.
//                                                                           
//  Disclaimer:                                                                           
//    This project is provided without any guarantee and can be used for   
//    private and commercial purposes. Any use is at the user’s 
//    own risk and responsibility.
//
// -------------------------------------------------------------------------
TYPE StepMode :
(
  /// StepMode is deactivated
  DEACTIVATE := 0,
  /// Blending
  /// • The robot moves on the blended trajectory
  /// • The movement is interrupted when the active segment changes
  BLENDING := 1,
  ///Exact stop
  /// • The robot moves to the defined target positions without blending
  /// • The movement is interrupted when the defined target position is reached
  EXACT_STOP := 2
)USINT;
END_TYPE

{attribute 'qualified_only'}
// ------------------------------------------------------------------------- 
//  SRCI Robot Library                                                
// ------------------------------------------------------------------------- 
//                                                                           
//  Object:      StopMode                                       
//  Author:      Thorsten Brach                                                
//  Date:        2024-06-01
//
//  Description:                                              
//   
//                                                                           
//  Copyright: 
//    (C) 2024 Thorsten Brach. All rights reserved                                                                                                                                            
//             Licensed under the MIT License.
//                                                                           
//  Disclaimer:                                                                           
//    This project is provided without any guarantee and can be used for   
//    private and commercial purposes. Any use is at the user’s 
//    own risk and responsibility.
//
// -------------------------------------------------------------------------
TYPE StopMode :
(
  /// 0: Stop via JobID (default)
  /// TargetID is interpreted as JobID
  /// All instances of the defined JobID are stopped
  STOP_JOB_ID := 0,  
  /// 1: Stop via InstanceID
  /// TargetID is interpreted as InstanceID
  /// The instance of the defined InstanceID is stopped
  STOP_INSTANCE_ID := 1,  
  /// 2: Stop all subprograms
  /// All subprograms independent of the input parameter value of TargetID are stopped
  STOP_ALL_SUBPROGRAMS := 2
)USINT;
END_TYPE

{attribute 'qualified_only'}
// ------------------------------------------------------------------------- 
//  SRCI Robot Library                                                
// ------------------------------------------------------------------------- 
//                                                                           
//  Object:      SyncInMode                                       
//  Author:      Thorsten Brach                                                
//  Date:        2024-06-01
//
//  Description:                                              
//   
//                                                                           
//  Copyright: 
//    (C) 2024 Thorsten Brach. All rights reserved                                                                                                                                            
//             Licensed under the MIT License.
//                                                                           
//  Disclaimer:                                                                           
//    This project is provided without any guarantee and can be used for   
//    private and commercial purposes. Any use is at the user’s 
//    own risk and responsibility.
//
// -------------------------------------------------------------------------
TYPE SyncInMode :
(
  /// • When work piece enters "SyncInZone"
  /// • Start synchronization as soon as possible within defined acceleration and velocity limits
  IN_SYNC_IN_ZONE := 0,
  /// • Start synchronization after specific distance after execution
  /// • "SynInZone" ignored
  AFTER_DISTANCE := 1,
  /// • Start synchronization after specific time after execution
  /// • "SynInZone" ignored
  AFTER_TIME := 2,
  /// • As soon as possible within defined acceleration and velocity limits
  /// • "SynInZone" ignored
  IMMEDIATELY := 3
)USINT;
END_TYPE

{attribute 'qualified_only'}
// ------------------------------------------------------------------------- 
//  SRCI Robot Library                                                
// ------------------------------------------------------------------------- 
//                                                                           
//  Object:      SyncMode                                       
//  Author:      Thorsten Brach                                                
//  Date:        2024-06-01
//
//  Description:                                              
//   
//                                                                           
//  Copyright: 
//    (C) 2024 Thorsten Brach. All rights reserved                                                                                                                                            
//             Licensed under the MIT License.
//                                                                           
//  Disclaimer:                                                                           
//    This project is provided without any guarantee and can be used for   
//    private and commercial purposes. Any use is at the user’s 
//    own risk and responsibility.
//
// -------------------------------------------------------------------------
TYPE SyncMode :
(
  /// No synchronization will be executed
  NO_SYNCHRONIZATION := 0,
  /// Server data will be overwritten immediately by client data
  CLIENT_TO_SERVER := 1,
  /// Client data will be overwritten immediately by server data
  SERVER_TO_CLIENT := 2,
  /// Server or client data will be overwritten immediately by changed data
  AUTOMATIC := 3
)USINT;
END_TYPE

{attribute 'qualified_only'}
// ------------------------------------------------------------------------- 
//  SRCI Robot Library                                                
// ------------------------------------------------------------------------- 
//                                                                           
//  Object:      ThresholdMode                                       
//  Author:      Thorsten Brach                                                
//  Date:        2024-06-01
//
//  Description:                                              
//   
//                                                                           
//  Copyright: 
//    (C) 2024 Thorsten Brach. All rights reserved                                                                                                                                            
//             Licensed under the MIT License.
//                                                                           
//  Disclaimer:                                                                           
//    This project is provided without any guarantee and can be used for   
//    private and commercial purposes. Any use is at the user’s 
//    own risk and responsibility.
//
// -------------------------------------------------------------------------
TYPE ThresholdMode :
(
  /// Automatic.
  AUTOMATIC := 0,
  /// Manual (according to LimitAxis)
  MANUAL    := 1
)USINT;
END_TYPE

{attribute 'qualified_only'}
// ------------------------------------------------------------------------- 
//  SRCI Robot Library                                                
// ------------------------------------------------------------------------- 
//                                                                           
//  Object:      ToolCalculationMode                                       
//  Author:      Thorsten Brach                                                
//  Date:        2024-06-01
//
//  Description:                                              
//   
//                                                                           
//  Copyright: 
//    (C) 2024 Thorsten Brach. All rights reserved                                                                                                                                            
//             Licensed under the MIT License.
//                                                                           
//  Disclaimer:                                                                           
//    This project is provided without any guarantee and can be used for   
//    private and commercial purposes. Any use is at the user’s 
//    own risk and responsibility.
//
// -------------------------------------------------------------------------
TYPE ToolCalculationMode :
(
  /// 0: Two Point + Z-Method (default)
  TWO_POINT_Z_METHOD := 0,        
  /// 1: Three-Point-Method
  THREE_POINT_METHOD := 1,        
  /// 2: Four-Point-Method
  FOUR_POINT_METHOD := 2,        
  /// 3: Five-Point-Method
  FIVE_POINT_METHOD := 3,        
  /// 4: Six-Point-Method
  SIX_POINT_METHOD := 4,        
  /// 5: ABC-World-Method
  ABC_WORLD_METHOD := 5,        
  /// 6: ABC-Two-Point-Method
  ABC_TWO_POINT_METHOD := 6
)SINT;
END_TYPE

{attribute 'qualified_only'}
// ------------------------------------------------------------------------- 
//  SRCI Robot Library                                                
// ------------------------------------------------------------------------- 
//                                                                           
//  Object:      TrajectoryMode                                       
//  Author:      Thorsten Brach                                                
//  Date:        2024-06-01
//
//  Description:                                              
//   
//                                                                           
//  Copyright: 
//    (C) 2024 Thorsten Brach. All rights reserved                                                                                                                                            
//             Licensed under the MIT License.
//                                                                           
//  Disclaimer:                                                                           
//    This project is provided without any guarantee and can be used for   
//    private and commercial purposes. Any use is at the user’s 
//    own risk and responsibility.
//
// -------------------------------------------------------------------------
TYPE TrajectoryMode :
(
  /// Invalid (default)
  INVALID := 0,
  /// Linear movement
  LINEAR_MOVEMENT := 1,
  /// PTP movement
  PTP_MOVEMENT := 2
)USINT;
END_TYPE

{attribute 'qualified_only'}
// ------------------------------------------------------------------------- 
//  SRCI Robot Library                                                
// ------------------------------------------------------------------------- 
//                                                                           
//  Object:      TransformMode                                       
//  Author:      Thorsten Brach                                                
//  Date:        2024-06-01
//
//  Description:                                              
//   
//                                                                           
//  Copyright: 
//    (C) 2024 Thorsten Brach. All rights reserved                                                                                                                                            
//             Licensed under the MIT License.
//                                                                           
//  Disclaimer:                                                                           
//    This project is provided without any guarantee and can be used for   
//    private and commercial purposes. Any use is at the user’s 
//    own risk and responsibility.
//
// -------------------------------------------------------------------------
TYPE TransformMode :
(
  /// 0 (default): Mirror at Point with mirroring of the target position’s orientation
  /// Requires for the mirror Point the "TransformationParameter_1" and the "TransformationParameter_2" set to "Not used"
  MIRROR_AT_POINT := 0,  
  /// 1: Mirror at Straight Line with mirroring of the target position’s orientation
  /// Requires for the Straight Line the "TransformationParameter_1" and the "TransformationParameter_2" set to "X-Axis", "Y-Axis" or "Z-Axis"
  MIRROR_AT_STRAIGHT_LINE := 1,  
  /// 2: Mirror at Plane with mirroring of the target position’s orientation
  /// Requires for the Plane the "TransformationParameter_1" and the "TransformationParameter_2" set to "XY-Axis", "XZ-Axis" or "YZ-Axis"
  MIRROR_AT_PLANE := 2,  
  /// 3: Rotate around Straight Line with rotation of the target position’s orientation
  /// Requires for the Straight Line the "TransformationParameter_1" and the "TransformationParameter_2" set to "X-Axis", "Y-Axis" or "Z-Axis"
  /// Requires for the parameter "RotationAngle"
  ROTATE_AROUND_STRAIGHT_LINE := 3,  
  /// 4: Shift by Vector
  /// Requires for the shifting Vector defined by the Point the "TransformationParameter_1" and the "TransformationParameter_2" set to "Not used"
  /// Requires for the shifting shortest Vector to the Straight Line the "TransformationParameter_1" and the "TransformationParameter_2" set to "X-Axis", "Y-Axis" or "Z-Axis"
  /// Requires for the shifting shortest Vector to the Plane the "TransformationParameter_1" and the "TransformationParameter_2" set to "XY-Axis", "XZ-Axis" or "YZ-Axis"
  SHIFT_BY_VECTOR := 4
)SINT;
END_TYPE

{attribute 'qualified_only'}
// ------------------------------------------------------------------------- 
//  SRCI Robot Library                                                
// ------------------------------------------------------------------------- 
//                                                                           
//  Object:      TriggerModeIo                                       
//  Author:      Thorsten Brach                                                
//  Date:        2024-06-01
//
//  Description:                                              
//   
//                                                                           
//  Copyright: 
//    C) 2024 Thorsten Brach. All rights reserved                                                                                                                                            
//             Licensed under the MIT License.
//                                                                           
//  Disclaimer:                                                                           
//    This project is provided without any guarantee and can be used for   
//    private and commercial purposes. Any use is at the user’s 
//    own risk and responsibility.
//
// -------------------------------------------------------------------------
TYPE TriggerModeIo :
(
  /// Invalid (default)
  INVALID := 0,  
  /// Digital Input Rising Edge
  DIGITAL_INPUT_RISING_EDGE := 10,
  /// Digital Input Falling Edge
  DIGITAL_INPUT_FALLING_EDGE := 11,
  /// Digital Input Rising or Falling Edge
  DIGITAL_INPUT_RISING_OR_FALLING_EDGE := 12,
  /// Digital Input Rising or Falling Edge (Inverted)
  DIGITAL_INPUT_RISING_OR_FALLING_EDGE_INVERTED := 13,
  /// Digital Output Rising Edge
  DIGITAL_OUTPUT_RISING_EDGE := 20,
  /// Digital Output Falling Edge
  DIGITAL_OUTPUT_FALLING_EDGE := 21,
  /// Digital Output Rising or Falling Edge
  DIGITAL_OUTPUT_RISING_OR_FALLING_EDGE := 22,
  /// Digital Output Rising or Falling Edge (Inverted)
  DIGITAL_OUTPUT_RISING_OR_FALLING_EDGE_INVERTED := 23,
  /// Analog Input Exceeding Defined Threshold
  ANALOG_INPUT_EXCEEDING_DEFINED_THRESHOLD := 30,
  /// Analog Input Falling Below Defined Threshold
  ANALOG_INPUT_FALLING_BELOW_DEFINED_THRESHOLD := 31,
  /// Analog Input Exceeding or Falling Below Defined Threshold
  ANALOG_INPUT_EXCEEDING_OR_FALLING_BELOW_DEFINED_THRESHOLD := 32,
  /// Analog Input Exceeding or Falling Below Defined Threshold (Inverted)
  ANALOG_INPUT_EXCEEDING_OR_FALLING_BELOW_DEFINED_THRESHOLD_INVERTED := 33,
  /// Analog Input Entering Defined Range
  ANALOG_INPUT_ENTERING_DEFINED_RANGE := 34,
  /// Analog Input Leaving Defined Range
  ANALOG_INPUT_LEAVING_DEFINED_RANGE := 35,
  /// Analog Input Entering or Leaving Defined Range
  ANALOG_INPUT_ENTERING_OR_LEAVING_DEFINED_RANGE := 36,
  /// Analog Input Entering or Leaving Defined Range (Inverted)
  ANALOG_INPUT_ENTERING_OR_LEAVING_DEFINED_RANGE_INVERTED := 37,
  /// Analog Output Exceeding Defined Threshold
  ANALOG_OUTPUT_EXCEEDING_DEFINED_THRESHOLD := 40,
  /// Analog Output Falling Below Defined Threshold
  ANALOG_OUTPUT_FALLING_BELOW_DEFINED_THRESHOLD := 41,
  /// Analog Output Exceeding or Falling Below Defined Threshold
  ANALOG_OUTPUT_EXCEEDING_OR_FALLING_BELOW_DEFINED_THRESHOLD := 42,
  /// Analog Output Exceeding or Falling Below Defined Threshold (Inverted)
  ANALOG_OUTPUT_EXCEEDING_OR_FALLING_BELOW_DEFINED_THRESHOLD_INVERTED := 43,
  /// Analog Output Entering Defined Range
  ANALOG_OUTPUT_ENTERING_DEFINED_RANGE := 44,
  /// Analog Output Leaving Defined Range
  ANALOG_OUTPUT_LEAVING_DEFINED_RANGE := 45,
  /// Analog Output Entering or Leaving Defined Range
  ANALOG_OUTPUT_ENTERING_OR_LEAVING_DEFINED_RANGE := 46,
  /// Analog Output Entering or Leaving Defined Range (Inverted)
  ANALOG_OUTPUT_ENTERING_OR_LEAVING_DEFINED_RANGE_INVERTED := 47,
  /// Integer Register Exceeding Defined Threshold
  INTEGER_REGISTER_EXCEEDING_DEFINED_THRESHOLD := 50,
  /// Integer Register Falling Below Defined Threshold
  INTEGER_REGISTER_FALLING_BELOW_DEFINED_THRESHOLD := 51,
  /// Integer Register Exceeding or Falling Below Defined Threshold
  INTEGER_REGISTER_EXCEEDING_OR_FALLING_BELOW_DEFINED_THRESHOLD := 52,
  /// Integer Register Exceeding or Falling Below Defined Value (Inverted)
  INTEGER_REGISTER_EXCEEDING_OR_FALLING_BELOW_DEFINED_VALUE_INVERTED := 53,
  /// Integer Register Entering Defined Range
  INTEGER_REGISTER_ENTERING_DEFINED_RANGE := 54,
  /// Integer Register Leaving Defined Range
  INTEGER_REGISTER_LEAVING_DEFINED_RANGE := 55,
  /// Integer Register Entering or Leaving Defined Range
  INTEGER_REGISTER_ENTERING_OR_LEAVING_DEFINED_RANGE := 56,
  /// Integer Register Entering or Leaving Defined Range (Inverted)
  INTEGER_REGISTER_ENTERING_OR_LEAVING_DEFINED_RANGE_INVERTED := 57,
  /// Real Register Exceeding Defined Threshold
  REAL_REGISTER_EXCEEDING_DEFINED_THRESHOLD := 60,
  /// Real Register Falling Below Defined Threshold
  REAL_REGISTER_FALLING_BELOW_DEFINED_THRESHOLD := 61,
  /// Real Register Exceeding or Falling Below Defined Threshold
  REAL_REGISTER_EXCEEDING_OR_FALLING_BELOW_DEFINED_THRESHOLD := 62,
  /// Real Register Exceeding or Falling Below Defined Threshold (Inverted)
  REAL_REGISTER_EXCEEDING_OR_FALLING_BELOW_DEFINED_THRESHOLD_INVERTED := 63,
  /// Real Register Entering Defined Range
  REAL_REGISTER_ENTERING_DEFINED_RANGE := 64,
  /// Real Register Leaving Defined Range
  REAL_REGISTER_LEAVING_DEFINED_RANGE := 65,
  /// Real Register Entering or Leaving Defined Range
  REAL_REGISTER_ENTERING_OR_LEAVING_DEFINED_RANGE := 66,
  /// Real Register Entering or Leaving Defined Range (Inverted)
  REAL_REGISTER_ENTERING_OR_LEAVING_DEFINED_RANGE_INVERTED := 67
)SINT;
END_TYPE

{attribute 'qualified_only'}
// ------------------------------------------------------------------------- 
//  SRCI Robot Library                                                
// ------------------------------------------------------------------------- 
//                                                                           
//  Object:      TriggerModeLimit                                       
//  Author:      Thorsten Brach                                                
//  Date:        2024-06-01
//
//  Description:                                              
//   
//                                                                           
//  Copyright: 
//    (C) 2024 Thorsten Brach. All rights reserved                                                                                                                                            
//             Licensed under the MIT License.
//                                                                           
//  Disclaimer:                                                                           
//    This project is provided without any guarantee and can be used for   
//    private and commercial purposes. Any use is at the user’s 
//    own risk and responsibility.
//
// -------------------------------------------------------------------------
TYPE TriggerModeLimit :
(
  /// 0: Invalid (default)
  INVALID := 0,
  /// 1: Joint current in mA
  JOINT_CURRENT := 1,
  /// 2: Force in Nm
  FORCE := 2,
  /// 3: Following error. The distance of the robot position from the path that was calculated
  FOLLOWING_ERROR := 3,
  /// Temperature in °C
  TEMPERATURE := 4  
)SINT;
END_TYPE

{attribute 'qualified_only'}
// ------------------------------------------------------------------------- 
//  SRCI Robot Library                                                
// ------------------------------------------------------------------------- 
//                                                                           
//  Object:      TriggerModeMeasurement                                       
//  Author:      Thorsten Brach                                                
//  Date:        2024-06-01
//
//  Description:                                              
//   
//                                                                           
//  Copyright: 
//    (C) 2024 Thorsten Brach. All rights reserved                                                                                                                                            
//             Licensed under the MIT License.
//                                                                           
//  Disclaimer:                                                                           
//    This project is provided without any guarantee and can be used for   
//    private and commercial purposes. Any use is at the user’s 
//    own risk and responsibility.
//
// -------------------------------------------------------------------------
TYPE TriggerModeMeasurement :
(
  /// (default) No trigger related behavior
  NO_TRIGGER := 0,
  /// 1: Starts the measurement with the positive trigger event and stops it with the negative trigger event 
  ///    when the trigger function with the identical EmitterID is activated.
  POSITIVE_START_NEGATIVE_STOP := 1,
  /// 2: Starts and stops the measurement with the positive trigger event 
  ///    when the trigger function with the identical EmitterID is activated.
  POSITIVE_START_STOP := 2
)USINT;
END_TYPE

{attribute 'qualified_only'}
// ------------------------------------------------------------------------- 
//  SRCI Robot Library                                                
// ------------------------------------------------------------------------- 
//                                                                           
//  Object:      TriggerReactionMode                                       
//  Author:      Thorsten Brach                                                
//  Date:        2024-06-01
//
//  Description:                                              
//   
//                                                                           
//  Copyright: 
//    (C) 2024 Thorsten Brach. All rights reserved                                                                                                                                            
//             Licensed under the MIT License.
//                                                                           
//  Disclaimer:                                                                           
//    This project is provided without any guarantee and can be used for   
//    private and commercial purposes. Any use is at the user’s 
//    own risk and responsibility.
//
// -------------------------------------------------------------------------
TYPE TriggerReactionMode :
(
/// No reaction (default).
  NO_REACTION := 0,
  /// Interrupt: Robot movement is paused. Movement can be continued by function GroupContinue.
  INTERRUPT := 1,
  /// GroupStop: Robot stops the movement and brings all axes to a halt. Movements aborted by this command cannot be continued.
  GROUP_STOP := 2,
  /// Disable robot: The robot’s drives are disabled. This leads to the robot state "Not enabled" (see chapter 5.5.3).
  DISABLE_ROBOT := 3,
  /// Stop actual motion command: Robot movement is paused. Movement can be continued by the next motion command.
  STOP_ACTUAL_MOTION_COMMAND := 4
)SINT;
END_TYPE

{attribute 'qualified_only'}
// ------------------------------------------------------------------------- 
//  SRCI Robot Library                                                
// ------------------------------------------------------------------------- 
//                                                                           
//  Object:      TurnMode                                       
//  Author:      Thorsten Brach                                                
//  Date:        2024-06-01
//
//  Description:                                              
//   
//                                                                           
//  Copyright: 
//    (C) 2024 Thorsten Brach. All rights reserved                                                                                                                                            
//             Licensed under the MIT License.
//                                                                           
//  Disclaimer:                                                                           
//    This project is provided without any guarantee and can be used for   
//    private and commercial purposes. Any use is at the user’s 
//    own risk and responsibility.
//
// -------------------------------------------------------------------------
TYPE TurnMode :
(
  /// Use TurnNumber in position
  USE_TURN_NUMBER := 0,
  ///  Do not change TurnNumber with this movement
  SAME            := 1,
  /// TurnNumber in position is not used but the Robot is free to change TurnNumber
  FREE            := 2
)USINT;
END_TYPE

{attribute 'qualified_only'}
// ------------------------------------------------------------------------- 
//  SRCI Robot Library                                                
// ------------------------------------------------------------------------- 
//                                                                           
//  Object:      WorkAreaReactionMode                                       
//  Author:      Thorsten Brach                                                
//  Date:        2024-06-01
//
//  Description:                                              
//   
//                                                                           
//  Copyright: 
//    (C) 2024 Thorsten Brach. All rights reserved                                                                                                                                            
//             Licensed under the MIT License.
//                                                                           
//  Disclaimer:                                                                           
//    This project is provided without any guarantee and can be used for   
//    private and commercial purposes. Any use is at the user’s 
//    own risk and responsibility.
//
// -------------------------------------------------------------------------
TYPE WorkAreaReactionMode :
(
  /// 0: No reaction (default)
  /// • RC reports violation
  /// • Robot is not stopped
  NO_REACTION := 0,
  /// 
  /// 1: Abort
  /// • RC reports violation
  /// • RC returns error
  /// • Robot is stopped
  /// • Sequence buffer emptied
  ABORT := 1,
  /// 2: Interrupt
  /// • RC reports violation
  /// • Robot movement is paused
  /// • Movement can be continued by function GroupContinue
   INTERRUPT := 2
)USINT;
END_TYPE

{attribute 'qualified_only'}
// ------------------------------------------------------------------------- 
//  SRCI Robot Library                                                
// ------------------------------------------------------------------------- 
//                                                                           
//  Object:      ActiveCommandRegisterState                                       
//  Author:      Thorsten Brach                                                
//  Date:        2024-06-01
//
//  Description:                                              
//   
//                                                                           
//  Copyright: 
//    (C) 2024 Thorsten Brach. All rights reserved                                                                                                                                            
//             Licensed under the MIT License.
//                                                                           
//  Disclaimer:                                                                           
//    This project is provided without any guarantee and can be used for   
//    private and commercial purposes. Any use is at the user’s 
//    own risk and responsibility.
//
// -------------------------------------------------------------------------
TYPE ActiveCommandRegisterState :
(
  /// IS_FREE denotes not used but available resources (empty slots in the ACR).
  IS_FREE        := 0,
  /// IS_PROCESSING CMDs are actively being processed by client or server. 
  /// In terms of CMD category, IS_PROCESSING also describes commands whose tasks are not currently being executed (not ACTIVE), 
  /// but e.g. a CMD waiting in the Sequence buffer.
  IS_PROCESSING := 1,
  /// IS_FINAL states are reached on CMD termination. Execution of this Task has been finished and its results can be examined.
  IS_FINAL    := 2
);
END_TYPE

{attribute 'qualified_only'}
// ------------------------------------------------------------------------- 
//  SRCI Robot Library                                                
// ------------------------------------------------------------------------- 
//                                                                           
//  Object:      BufferStateCmd                                       
//  Author:      Thorsten Brach                                                
//  Date:        2024-06-01
//
//  Description:                                              
//   
//                                                                           
//  Copyright: 
//    (C) 2024 Thorsten Brach. All rights reserved                                                                                                                                            
//             Licensed under the MIT License.
//                                                                           
//  Disclaimer:                                                                           
//    This project is provided without any guarantee and can be used for   
//    private and commercial purposes. Any use is at the user’s 
//    own risk and responsibility.
//
// -------------------------------------------------------------------------
TYPE BufferStateCmd :
(
 // PDF Page 353 
  EMPTY            := 0,
  CREATED          := 1,
  UPDATE_AVAILABLE := 2,
  SENDING          := 3,
  PROCESSED        := 4  
);
END_TYPE

{attribute 'qualified_only'}
// ------------------------------------------------------------------------- 
//  SRCI Robot Library                                                
// ------------------------------------------------------------------------- 
//                                                                           
//  Object:      BufferStateRsp                                       
//  Author:      Thorsten Brach                                                
//  Date:        2024-06-01
//
//  Description:                                              
//   
//                                                                           
//  Copyright: 
//    (C) 2024 Thorsten Brach. All rights reserved                                                                                                                                            
//             Licensed under the MIT License.
//                                                                           
//  Disclaimer:                                                                           
//    This project is provided without any guarantee and can be used for   
//    private and commercial purposes. Any use is at the user’s 
//    own risk and responsibility.
//
// -------------------------------------------------------------------------
TYPE BufferStateRsp :
(
 // PDF Seite 353 
  EMPTY            := 0,
  RECEIVING        := 1,
  RECEIVED         := 2,
  PROCESSED        := 3  
);
END_TYPE

{attribute 'qualified_only'}
// ------------------------------------------------------------------------- 
//  SRCI Robot Library                                                
// ------------------------------------------------------------------------- 
//                                                                           
//  Object:      CmdMessageState                                       
//  Author:      Thorsten Brach                                                
//  Date:        2024-06-01
//
//  Description:                                              
//   
//                                                                           
//  Copyright: 
//    (C) 2024 Thorsten Brach. All rights reserved                                                                                                                                            
//             Licensed under the MIT License.
//                                                                           
//  Disclaimer:                                                                           
//    This project is provided without any guarantee and can be used for   
//    private and commercial purposes. Any use is at the user’s 
//    own risk and responsibility.
//
// -------------------------------------------------------------------------
TYPE CmdMessageState :
(
  /// No operation or process is active
  EMPTY := 0,
  /// Created but not yet started
  CREATED := 1,
  /// Buffered and awaiting execution
  BUFFERED := 2,
  /// Buffered in planner for future execution
  BUFFERED_IN_PLANNER := 3,
  /// Currently active and in progress
  ACTIVE := 4,
  /// Interrupted and awaiting continuation
  INTERRUPTED := 5,
  /// Requested for abort
  ABORT_REQUEST := 6,
  /// Successfully completed
  DONE := 10,
  /// Aborted before completion
  ABORTED := 14,
  /// Encountered an error during execution
  ERROR := 15
)USINT;
END_TYPE

{attribute 'qualified_only'}
// ------------------------------------------------------------------------- 
//  SRCI Robot Library                                                
// ------------------------------------------------------------------------- 
//                                                                           
//  Object:      InitializationState                                       
//  Author:      Thorsten Brach                                                
//  Date:        2024-06-01
//
//  Description:                                              
//   
//                                                                           
//  Copyright: 
//    (C) 2024 Thorsten Brach. All rights reserved                                                                                                                                            
//             Licensed under the MIT License.
//                                                                           
//  Disclaimer:                                                                           
//    This project is provided without any guarantee and can be used for   
//    private and commercial purposes. Any use is at the user’s 
//    own risk and responsibility.
//
// -------------------------------------------------------------------------
TYPE InitializationState :
(
  /// Default
  DEFAULT := 0,
  /// Error: Telegram control does not match the telegram state
  ERROR_TELEGRAM_CONTROL := 161,
  /// Error: Initialization lost for unknown reason. See message log after reinitializing
  ERROR_INIT_LOST := 162,
  /// Error: Telegram length does not match the length provided in the communication interface.
  ERROR_TELEGRAM_LENGTH := 163,
  /// Error: Incompatible major SRCI version
  ERROR_INCOMPATIBLE_SRCI := 164,
  /// Error: Lifesign timeout
  ERROR_LIFESIGN_TIMEOUT := 165,
  /// Error: The selected optional cyclic data does not fit in the given telegram size
  ERROR_CYCLIC_DATA_MISMATCH := 166,
  /// Error: The robot interface was reset after being initialized
  ERROR_INTERFACE_RESET := 167,
  /// Error: Telegram sequence timeout
  ERROR_SEQUENCE_TIMEOUT := 168,
  /// Error: The telegram number changed after initialization
  ERROR_TELEGRAM_NUMBER_CHANGED := 169,
  /// Error: Invalid AxesGroupID
  ERROR_INVALID_AXES_GROUP := 170,
  /// Error: Telegram number is invalid. E.g. TwoSequences is only activated in one direction
  ERROR_INVALID_TELEGRAM_NUMBER := 171,
  /// Error: Telegram Number is not supported
  ERROR_TELEGRAM_NUMBER_NOT_SUPPORTED := 172,
  /// Ready to resume: The RC is currently not initialized but has state in the ACR
  READY_TO_RESUME := 253,
  /// Ready for initialization: The RC is currently not initialized and has no state in the ACR
  READY_FOR_INITIALIZATION := 254,
  /// Initialized: The RC state is Initialized
  INITIALIZED := 255
);
END_TYPE

{attribute 'qualified_only'}
// ------------------------------------------------------------------------- 
//  SRCI Robot Library                                                
// ------------------------------------------------------------------------- 
//                                                                           
//  Object:      RaPowerState                                       
//  Author:      Thorsten Brach                                                
//  Date:        2024-06-01
//
//  Description:                                              
//   
//                                                                           
//  Copyright: 
//    (C) 2024 Thorsten Brach. All rights reserved                                                                                                                                            
//             Licensed under the MIT License.
//                                                                           
//  Disclaimer:                                                                           
//    This project is provided without any guarantee and can be used for   
//    private and commercial purposes. Any use is at the user’s 
//    own risk and responsibility.
//
// -------------------------------------------------------------------------
TYPE RaPowerState :
(
  /// Robot drives disabled. Robot cannot be moved
  NOT_ENABLED := 0,
  /// Robot drives powered on. Robot can be moved according to sequence state
  ENABLED := 1
)USINT;
END_TYPE

{attribute 'qualified_only'}
// ------------------------------------------------------------------------- 
//  SRCI Robot Library                                                
// ------------------------------------------------------------------------- 
//                                                                           
//  Object:      RaSequenceState                                       
//  Author:      Thorsten Brach                                                
//  Date:        2024-06-01
//
//  Description:                                              
//   
//                                                                           
//  Copyright: 
//    (C) 2024 Thorsten Brach. All rights reserved                                                                                                                                            
//             Licensed under the MIT License.
//                                                                           
//  Disclaimer:                                                                           
//    This project is provided without any guarantee and can be used for   
//    private and commercial purposes. Any use is at the user’s 
//    own risk and responsibility.
//
// -------------------------------------------------------------------------
TYPE RaSequenceState :
(
  /// Robot can be moved by incoming command
  IDLE := 0,
  /// RC is processing command in active sequence
  EXECUTING := 1,
  /// Interrupt is active. Robot is waiting for Continue
  INTERRUPTED := 2
)USINT;
END_TYPE

